PROGRAM MAIN
VAR
	testMover : Mover;
END_VAR

testMover.CyclicLogic();

END_PROGRAM

(* stored: Version 1.1.0.1
   POU MAIN: Id {8e9720ae-ba12-41bf-b205-4bd149d86cd8}, SpecialFunc None *)
